PROGRAM P_Foldedoer_4_213
(*
Rummene er delt af en foldedør med dørkontakt i rum 4.213. Når dørkontakt aktiveres behandles de to rum som ét rum:
	- Senorinput sammensættes, således de to reguleringer har samme PV.
	- Knapfunktion sammensættes, således alle knapper kan benyttes for hele rummet.
Sammensætning af sensorinput foregår i FB_FoldingDoor.A_SensorLogic (SH_Light)
Sammensætning af knapfunktion foregår i FB_FoldingDoor.A_ButtonLogic (SH_Light)

Rækkefølge i arrays: [1, 2] = [*rum 4.213*, *rum 4.215*]
*)
VAR
	bFoldingDoorOpen 		AT %I*	: BOOL;
	
	arrTopButtonZone1						: ARRAY[1..2] OF BOOL; //Fra GVL_EnOcean
	arrBottomButtonZone1					: ARRAY[1..2] OF BOOL; //Fra GVL_EnOcean
	arrTopButtonZone1Comb				: ARRAY[1..2] OF BOOL; //Til A_Buttons
	arrBottomButtonZone1Comb			: ARRAY[1..2] OF BOOL; //Til A_Buttons
	
	arrstPirSensorData						: ARRAY[1..2] OF SH_Light.ST_DALI_Sensor; //VAR_IN_OUT til og fra sensorer
	arrstPirSensorDataComb				: ARRAY[1..2] OF SH_Light.ST_DALI_Sensor; //VAR_IN_OUT til og fra LightCtrl
	
	fbFoldingDoor								: SH_Light.FB_FoldingDoor;
END_VAR

arrTopButtonZone1[1]		:= GVL_EnOcean.strEnOceanSwitch_Rum_4_213_Indgang.bT2_ON;
arrBottomButtonZone1[1]	:= GVL_EnOcean.strEnOceanSwitch_Rum_4_213_Indgang.bT2_OFF;
arrTopButtonZone1[2]		:= GVL_EnOcean.strEnOceanSwitch_Rum_4_215.bT2_ON;
arrBottomButtonZone1[2]	:= GVL_EnOcean.strEnOceanSwitch_Rum_4_215.bT2_OFF;

fbFoldingDoor(
	bFoldingDoorOpen 				:= bFoldingDoorOpen,
	arrTopButtonZone1 				:= arrTopButtonZone1,
	arrBottomButtonZone1			:= arrBottomButtonZone1,
	arrstPirSensorData				:= arrstPirSensorData,
	arrstPirSensorDataComb		:= arrstPirSensorDataComb,
	arrTopButtonZone1Comb		=> arrTopButtonZone1Comb,
	arrBottomButtonZone1Comb	=> arrBottomButtonZone1Comb);
(*
A_ButtonLogic();
A_SensorLogic();
*)

ACTION A_ButtonLogic:
arrTopButtonZone1[1] := GVL_EnOcean.strEnOceanSwitch_Rum_4_217.bT2_OFF;
arrBottomButtonZone1[1] := GVL_EnOcean.strEnOceanSwitch_Rum_4_217.bT2_ON;
arrTopButtonZone1[2] := GVL_EnOcean.strEnOceanSwitch_Rum_4_219.bT2_ON;
arrBottomButtonZone1[2] := GVL_EnOcean.strEnOceanSwitch_Rum_4_219.bT2_OFF;

IF bFoldingDoorOpen THEN
	arrTopButtonZone1Comb[1] := arrTopButtonZone1[1] OR arrTopButtonZone1[2];
	arrTopButtonZone1Comb[2] := arrTopButtonZone1Comb[1];
	arrBottomButtonZone1Comb[1] := arrBottomButtonZone1[1] OR arrBottomButtonZone1[2];
	arrBottomButtonZone1Comb[2] := arrBottomButtonZone1Comb[1];
ELSE
	arrTopButtonZone1Comb := arrTopButtonZone1;
	arrBottomButtonZone1Comb := arrBottomButtonZone1;
END_IF
END_ACTION

ACTION A_SensorLogic:
IF bFoldingDoorOpen THEN
	//Input fra sensorer samles
	arrstPirSensorDataComb[1].fBrightness			:= MIN(arrstPirSensorData[1].fBrightness, arrstPirSensorData[2].fBrightness);
	arrstPirSensorDataComb[1].bPrc					:= arrstPirSensorData[1].bPrc OR arrstPirSensorData[2].bPrc;
	arrstPirSensorDataComb[1].bBrightnessRead	:= arrstPirSensorData[1].bBrightnessRead OR arrstPirSensorData[2].bBrightnessRead;
	arrstPirSensorDataComb[2].fBrightness			:= arrstPirSensorDataComb[1].fBrightness;
	arrstPirSensorDataComb[2].bPrc					:= arrstPirSensorDataComb[1].bPrc;
	arrstPirSensorDataComb[2].bBrightnessRead	:= arrstPirSensorDataComb[1].bBrightnessRead;

	//Output til sensorer fordeles
	IF arrstPirSensorDataComb[1].bQueryBrightness OR arrstPirSensorDataComb[2].bQueryBrightness THEN
		arrstPirSensorData[1].bQueryBrightness := TRUE;
		arrstPirSensorData[2].bQueryBrightness := TRUE;
	ELSE
		arrstPirSensorData[1].bQueryBrightness := FALSE;
		arrstPirSensorData[2].bQueryBrightness := FALSE;
	END_IF
ELSE
	//Input fra sensorer samles uden ændring
	arrstPirSensorDataComb[1].fBrightness			:= arrstPirSensorData[1].fBrightness;
	arrstPirSensorDataComb[1].bPrc					:= arrstPirSensorData[1].bPrc;
	arrstPirSensorDataComb[1].bBrightnessRead	:= arrstPirSensorData[1].bBrightnessRead;
	arrstPirSensorDataComb[2].fBrightness			:= arrstPirSensorData[2].fBrightness;
	arrstPirSensorDataComb[2].bPrc					:= arrstPirSensorData[2].bPrc;
	arrstPirSensorDataComb[2].bBrightnessRead := arrstPirSensorData[2].bBrightnessRead;
	
	//Output til sensorer fordeles uden ændring
	IF arrstPirSensorDataComb[1].bQueryBrightness THEN
		arrstPirSensorData[1].bQueryBrightness := TRUE;
	ELSE
		arrstPirSensorData[1].bQueryBrightness := FALSE;
	END_IF
	IF arrstPirSensorDataComb[2].bQueryBrightness THEN
		arrstPirSensorData[2].bQueryBrightness := TRUE;
	ELSE
		arrstPirSensorData[2].bQueryBrightness := FALSE;
	END_IF
END_IF
END_ACTION

END_PROGRAM

(* stored: Version 1.1.0.1
   POU P_Foldedoer_4_213: Id {113bd217-ebc1-4194-8590-ae4936340b75}, SpecialFunc None
   Action A_ButtonLogic: Id {f5341b51-aaf5-470d-a876-403532d7bbde}
   Action A_SensorLogic: Id {ed4afc4c-58c6-45bb-89c4-01fbf9eaf428} *)
